(* CODESYS project Flags.library
   Company: _
   DefaultNamespace: Flags
   Title: Flags
   Placeholder: _Flags
   Author: Krystian Lis et al.
   Description: Boolean flags to share between domains.
   Version: 1.0.0

Project tree, tasks and I/O mapping:
  libraries: Debug, * (_); Results, * (_); Strings, * (_); Tags, * (_); Utils, * (_); Tc2_Standard, * (Beckhoff Automation GmbH); Tc2_System, * (Beckhoff Automation GmbH)
  Flag/
    Find/
      function FindFlag [ST]
      function FindManyFlags [ST]
      function FindWcdFlag [ST]
    Flag/
      function block A_Flag [ST]: FB_init
      global variables CFLAG
      function block Flag [ST]: FB_init, IsLowered, IsRised, Lower, Rise, Tag
      interface I_Flag: IsLowered, IsRised, Tag
    List/
      function block FlagList [ST]: _GetByTagIfTagged, _GetByTagIfUntagged, GetByPos, GetByTag, GetExtender, Release, Cap, IsReleased, Length, _ExtendIfTagged, _ExtendIfUntagged, _ExtendIfUntaggedIfNotEmpty, _PushIfTagged, _PushIfUntagged, Extend, Push
      function block FlagListExtender [ST]: List
      interface I_FlagList: GetByPos, GetByTag, GetExtender, Release, Cap, IsReleased, Length
      interface I_MutFlagList: Extend, Push
*)

// Flag/Flag/CFLAG
{attribute 'qualified_only'}
VAR_GLOBAL CONSTANT
	RISED		: Strings.Str := 'Rised';
	LOWERED		: Strings.Str := 'Lowered';
END_VAR

// Flag/Find/FindFlag
FUNCTION FindFlag : Results.Result
VAR_INPUT
	iFlagList		: I_FlagList;
	sToFind			: Strings.Str;
END_VAR
VAR_OUTPUT
	iFlag			: I_Flag;
END_VAR
VAR
	i			: Utils.GenIter(0);
	cmp			: Tags.TagCmp;
END_VAR

IF iFlagList = 0 THEN
	FindFlag := Results.Err.Itf0;
	RETURN;
END_IF

WHILE Results.IsOk(iFlagList.GetByPos(i.Next(), iFlag => iFlag)) DO
	IF cmp.Set(iFlag.Tag).MatchId(sToFind).IsTrue() THEN
		FindFlag := Results.Ok;
		RETURN;
	END_IF
END_WHILE

FindFlag := Results.Err.NoMatch;

END_FUNCTION

// Flag/List/I_FlagList
INTERFACE I_FlagList EXTENDS Debug.I_Debug

METHOD GetByPos : Results.Result
VAR_INPUT
	nPos			: UDINT;
END_VAR
VAR_OUTPUT
	iFlag			: I_Flag;
END_VAR
END_METHOD

METHOD GetByTag : Results.Result
VAR_INPUT
	iTag			: Tags.I_Tag;
END_VAR
VAR_OUTPUT
	iFlag			: I_Flag;
	nPos			: UDINT;
END_VAR
END_METHOD

METHOD GetExtender : FlagListExtender
VAR_INPUT
END_VAR
END_METHOD

METHOD Release : FlagListExtender;
END_METHOD

METHOD Cap : UDINT
VAR_INPUT
END_VAR
END_METHOD

METHOD IsReleased : BOOL
VAR_INPUT
END_VAR
END_METHOD

METHOD Length : UDINT
VAR_INPUT
END_VAR
END_METHOD

END_INTERFACE

// Flag/Flag/I_Flag
INTERFACE I_Flag EXTENDS Debug.I_Debug, Tags.I_Tagged

METHOD IsLowered : BOOL
VAR_INPUT
END_VAR
END_METHOD

METHOD IsRised : BOOL
VAR_INPUT
END_VAR
END_METHOD

PROPERTY Tag : Tags.I_Tag
GET
END_GET
END_PROPERTY

END_INTERFACE

// Flag/List/FlagListExtender
FUNCTION_BLOCK INTERNAL FlagListExtender
VAR
	_iList		: I_FlagList;
END_VAR

PROPERTY INTERNAL List : I_FlagList
GET
List := _iList;
END_GET
SET
_iList := List;
END_SET
END_PROPERTY

END_FUNCTION_BLOCK

// Flag/Find/FindManyFlags
FUNCTION FindManyFlags : Results.Result
VAR_INPUT
	iFlagList		: I_FlagList;
	nResultPou		: ANY;
END_VAR
VAR_IN_OUT
	sToFind		: ARRAY[*] OF Strings.Str;
END_VAR
VAR
	i			: Utils.GenIter(0);
	j			: UDINT;
	cmp			: Tags.TagCmp;
	_iFlag		: I_Flag;
	_nLow		: UDINT := DINT_TO_UDINT(LOWER_BOUND(sToFind, 1));
	_nUp		: UDINT := DINT_TO_UDINT(UPPER_BOUND(sToFind, 1));
	_nResSize	: UDINT := DINT_TO_UDINT(nResultPou.diSize);
	_nExpLen	: UDINT := _nUp - _nLow + 1;
	_nExpSize	: UDINT := _nExpLen * SIZEOF(__UXINT);
	
	_nFound		: UDINT := 0;
END_VAR

IF iFlagList = 0 THEN
	FindManyFlags := Results.Err.Itf0;
	RETURN;
END_IF

// Ensure lower bound starts at zero
IF _nLow <> 0 THEN
	FindManyFlags := Results.Err.Ovf;
	RETURN;
END_IF

// Ensure result size matches expected size
IF _nResSize <> _nExpSize THEN
	FindManyFlags := Results.Err.NoMatch;
	RETURN;
END_IF

// Check if result pointer is null
IF nResultPou.pValue = 0 THEN
	FindManyFlags := Results.Err.Ptr0;
	RETURN;
END_IF

// Iterate over the flag list
WHILE Results.IsOk(iFlagList.GetByPos(i.Next(), iFlag => _iFlag)) DO
	cmp.Set(_iFlag.Tag);
	FOR j := _nLow TO _nUp DO
		// Match the string and copy if successful
		IF cmp.MatchId(sToFind[j]).IsTrue() THEN
			Tc2_System.MEMCPY(ADR(nResultPou.pValue) + SIZEOF(__UXINT) * j, ADR(_iFlag), SIZEOF(__UXINT));
			_nFound := _nFound + 1;
			sToFind[j] := '';  // Mark as found
			EXIT;  // Break after first match (since there should be only one)
		END_IF
	END_FOR;
	
	// Early exit if all entries are found (this condition can be removed if only one flag is expected)
	IF _nFound = (_nUp - _nLow + 1) THEN
		FindManyFlags := Results.Ok;
		RETURN;
	END_IF 
END_WHILE

// Final check to see if all entries were processed
FOR j := _nLow TO _nUp DO
	IF sToFind[j] <> '' THEN  // Check for unfound entries
		FindManyFlags := Results.Err.Udf;  // Error if any remain unfound (handled at higher level)
		RETURN;
	END_IF
END_FOR

// Return success if everything is found
FindManyFlags := Results.Ok;

END_FUNCTION

// Flag/Flag/Flag
FUNCTION_BLOCK Flag IMPLEMENTS I_Flag
VAR
	_fbTag				: Tags.Tag;
	_bState				: BOOL;
END_VAR

//FB_Init is always available implicitly and it is used primarily for initialization.
//The return value is not evaluated. For a specific influence, you can also declare the
//methods explicitly and provide additional code there with the standard initialization
//code. You can evaluate the return value.
METHOD FB_Init: BOOL
VAR_INPUT
    bInitRetains: BOOL; // TRUE: the retain variables are initialized (reset warm / reset cold)
    bInCopyCode: BOOL;  // TRUE: the instance will be copied to the copy code afterward (online change)  
END_VAR
_fbTag.Option := CFLAG.LOWERED;
END_METHOD

METHOD IsLowered : BOOL
VAR_INPUT
END_VAR
IsLowered := _bState = FALSE;
END_METHOD

METHOD IsRised : BOOL
VAR_INPUT
END_VAR
IsRised := _bState = TRUE;
END_METHOD

METHOD Lower : BOOL
VAR_INPUT
END_VAR
_bState := FALSE;
_fbTag.Option := CFLAG.LOWERED;
END_METHOD

METHOD Rise : BOOL
VAR_INPUT
END_VAR
_bState := TRUE;
_fbTag.Option := CFLAG.RISED;
END_METHOD

PROPERTY Tag : Tags.I_Tag
GET
Tag := _fbTag;
END_GET
END_PROPERTY

END_FUNCTION_BLOCK

// Flag/Find/FindWcdFlag
FUNCTION FindWcdFlag : Results.Result
VAR_INPUT
	iFlagList		: I_FlagList;
	sToFind			: Strings.Str;
END_VAR
VAR_OUTPUT
	iFlag			: I_Flag;
END_VAR
VAR
	i			: Utils.GenIter(0);
	cmp			: Tags.TagCmp;
END_VAR

IF iFlagList = 0 THEN
	FindWcdFlag := Results.Err.Itf0;
	RETURN;
END_IF

WHILE Results.IsOk(iFlagList.GetByPos(i.Next(), iFlag => iFlag)) DO
	IF cmp.Set(iFlag.Tag).MatchWcdId(sToFind).IsTrue() THEN
		FindWcdFlag := Results.Ok;
		RETURN;
	END_IF
END_WHILE

FindWcdFlag := Results.Err.NoMatch;

END_FUNCTION

// Flag/Flag/A_Flag
FUNCTION_BLOCK A_Flag IMPLEMENTS Debug.I_Debug;

//FB_Init is always available implicitly and it is used primarily for initialization.
//The return value is not evaluated. For a specific influence, you can also declare the
//methods explicitly and provide additional code there with the standard initialization
//code. You can evaluate the return value.
METHOD FB_Init: BOOL
VAR_INPUT
    bInitRetains: BOOL; // TRUE: the retain variables are initialized (reset warm / reset cold)
    bInCopyCode: BOOL;  // TRUE: the instance will be copied to the copy code afterward (online change)
	iFlagList				: I_MutFlagList;
	iFlag					: I_Flag;
END_VAR
IF iFlagList = 0 THEN
	Debug.DebugMsg(THIS^, ': iFlagList: Itf = 0!');
	RETURN;
END_IF
IF iFlag = 0 THEN
	Debug.DebugMsg(THIS^, ': iFlag: Itf = 0!');
	RETURN;
END_IF

CASE iFlagList.Push(iFlag) OF
	Results.Ok:
		// No Error
	Results.None:
		Debug.DebugMsg(iFlagList, Tc2_Standard.CONCAT(__POUNAME(), ': Tried to insert a double!'));
		Debug.DebugMsg(iFlag, 'Im a double!');
	Results.Err.Ovf:
		Debug.DebugMsg(iFlagList, Tc2_Standard.CONCAT(__POUNAME(), ': Overflow!'));
		Debug.DebugMsg(iFlag, 'Cause of overflow!');
	Results.Err.NoMatch:
		Debug.DebugMsg(iFlagList, Tc2_Standard.CONCAT(__POUNAME(), ': No Match!'));
		Debug.DebugMsg(iFlag, 'This already have an owner!');
	ELSE
		Debug.DebugMsg(iFlagList, Tc2_Standard.CONCAT(__POUNAME(), ': Unknown Error!'));
		Debug.DebugMsg(iFlag, 'Cause!');		
END_CASE
END_METHOD

END_FUNCTION_BLOCK

// Flag/List/I_MutFlagList
INTERFACE I_MutFlagList EXTENDS Debug.I_Debug, I_FlagList

METHOD Extend 			: Results.Result
VAR_INPUT
	fbFlagListExtend	: FlagListExtender;
END_VAR
END_METHOD

METHOD Push : Results.Result
VAR_INPUT
	iFlag			: I_Flag;
END_VAR
VAR_OUTPUT
	nPos			: UDINT;
END_VAR
END_METHOD

END_INTERFACE

// Flag/List/FlagList
FUNCTION_BLOCK FlagList
VAR_GENERIC CONSTANT
	nMax				: UDINT(0..16#FFFFFFE) := 1;
END_VAR
IMPLEMENTS I_FlagList, I_MutFlagList
VAR
	_bIsReleased		: BOOL;
	_iFlag				: ARRAY[0..nMax] OF I_Flag;
	_nLen				: UDINT;
	_fbTagOwner			: Tags.TagOwner;
END_VAR

METHOD PRIVATE _GetByTagIfTagged : Results.Result
VAR_INPUT
	iTag				: Tags.I_Tag;
END_VAR
VAR_OUTPUT
	iFlag				: I_Flag;
	nPos				: UDINT;
END_VAR
IF iTag.Owner <> _fbTagOwner.Self THEN
	_GetByTagIfTagged := Results.None;
	RETURN;
END_IF

iFlag := _iFlag[iTag.Cache];
_GetByTagIfTagged := Results.Ok;
nPos := iTag.Cache;
END_METHOD

METHOD PRIVATE _GetByTagIfUntagged : Results.Result
VAR_INPUT
	iTag				: Tags.I_Tag;
END_VAR
VAR_OUTPUT
	iFlag				: I_Flag;
	nPos				: UDINT;
END_VAR
VAR
	i					: UDINT;
	cmp					: Tags.TagCmp;
END_VAR
FOR i := 0 TO _nLen - 1 DO
	IF cmp.Set(iTag).Match(_iFlag[i].Tag).IsTrue() THEN
		_GetByTagIfUntagged := Results.Ok;
		RETURN;
	END_IF	
END_FOR
END_METHOD

METHOD GetByPos : Results.Result
VAR_INPUT
	nPos		: UDINT;
END_VAR
VAR_OUTPUT
	iFlag		: I_Flag;
END_VAR
IF nPos > nMax THEN
	GetByPos := Results.Err.Ovf;
	RETURN;
END_IF

iFlag := _iFlag[nPos];
IF iFlag <> 0 THEN
	GetByPos := Results.Ok;
END_IF
END_METHOD

METHOD GetByTag : Results.Result;
VAR_INPUT
	iTag				: Tags.I_Tag;
END_VAR
VAR_OUTPUT
	iFlag				: I_Flag;
	nPos				: UDINT;
END_VAR
IF _nLen = 0 THEN
	GetByTag := Results.None;
	RETURN;
END_IF

IF iTag = 0 THEN
	GetByTag := Results.Err.Itf0;
	RETURN;
END_IF

IF _bIsReleased THEN
	GetByTag := _GetByTagIfUntagged(iTag, iFlag => iFlag, nPos => nPos);
ELSE
	GetByTag := _GetByTagIfTagged(iTag, iFlag => iFlag, nPos => nPos);
END_IF
END_METHOD

METHOD GetExtender : FlagListExtender
VAR_INPUT
END_VAR
GetExtender.List := THIS^;
END_METHOD

METHOD Release 				: FlagListExtender;
VAR
	i						: UDINT;
END_VAR
IF NOT _bIsReleased THEN
	FOR i := 0 TO _nLen - 1 DO
		_iFlag[i].Tag.Leave(_fbTagOwner);
	END_FOR
	
	_bIsReleased := TRUE;
END_IF

Release.List := THIS^;
END_METHOD

METHOD Cap : UDINT
VAR_INPUT
END_VAR
Cap := nMax;
END_METHOD

METHOD IsReleased : BOOL
VAR_INPUT
END_VAR
IsReleased := _bIsReleased;
END_METHOD

METHOD Length : UDINT
VAR_INPUT
END_VAR
Length := _nLen;
END_METHOD

METHOD PRIVATE _ExtendIfTagged : Results.Result
VAR_INPUT
	iFlagList			: I_FlagList;
END_VAR
VAR
	i					: UDINT;
	_iExtFlag			: I_Flag;
END_VAR
IF NOT iFlagList.IsReleased() THEN
	_ExtendIfTagged := Results.Err.NoMatch;
	RETURN;
END_IF

IF iFlagList.Length() + _nLen > nMax THEN
	_ExtendIfTagged := Results.Err.Ovf;
	RETURN;
END_IF

WHILE Results.IsOk(iFlagList.GetByPos(i, iFlag => _iExtFlag)) DO
	i := i + 1;
	_iExtFlag.Tag.Join(_fbTagOwner, _nLen);
	_iFlag[_nLen] := _iExtFlag;
	_nLen := _nLen + 1;
END_WHILE

_ExtendIfTagged := Results.Ok;
END_METHOD

METHOD PRIVATE _ExtendIfUntagged : Results.Result
VAR_INPUT
	iFlagList			: I_FlagList;
END_VAR
VAR
	i					: UDINT;
	j					: UDINT;

	_iExtFlag			: I_Flag;
	
END_VAR
IF _nLen <> 0 THEN
	_ExtendIfUntagged := _ExtendIfUntaggedIfNotEmpty(iFlagList);
ELSE
	IF iFlagList.Cap() > nMax THEN
		_ExtendIfUntagged := Results.Err.Ovf;
		RETURN;
	END_IF	

	WHILE Results.IsOk(iFlagList.GetByPos(i, iFlag => _iExtFlag)) DO
		i := i + 1;
		_iExtFlag.Tag.Join(_fbTagOwner, _nLen);
		_iFlag[_nLen] := _iExtFlag;
		_nLen := _nLen + 1;
	END_WHILE
	
	_ExtendIfUntagged := Results.Ok;
END_IF
END_METHOD

METHOD PRIVATE _ExtendIfUntaggedIfNotEmpty : Results.Result
VAR_INPUT
	iFlagList			: I_FlagList;
END_VAR
VAR
	i					: UDINT;
	j					: UDINT;
	k					: UDINT;

	_iTemp				: ARRAY[0..nMax] OF I_Flag;

	_nExtLen			: UDINT;
	_iExtFlag			: I_Flag;
END_VAR
WHILE Results.IsOk(iFlagList.GetByPos(i, iFlag => _iExtFlag)) DO
	
	FOR j := 0 TO _nLen - 1 DO
		IF _iFlag[j] = _iExtFlag THEN
			_iExtFlag := 0;
			EXIT;
		END_IF	
	END_FOR
	
	IF _iExtFlag <> 0 THEN
		_iTemp[k] := _iExtFlag;
		k := k + 1;
	END_IF
	
	i := i + 1;
END_WHILE

IF k = 0 THEN
	_ExtendIfUntaggedIfNotEmpty := Results.Ok;
	RETURN;
END_IF

FOR i := 0 TO k - 1 DO
	_iFlag[_nLen] := _iTemp[i];
	_nLen := _nLen + 1;
END_FOR

_ExtendIfUntaggedIfNotEmpty := Results.Ok;
END_METHOD

METHOD PRIVATE _PushIfTagged : Results.Result
VAR_INPUT
	iFlag			: I_Flag;
END_VAR
VAR_OUTPUT
	nPos			: UDINT;
END_VAR
VAR
	_iTag			: Tags.I_Tag;
END_VAR
IF iFlag = 0 THEN
	_PushIfTagged := Results.Err.Itf0;
	RETURN;
END_IF

IF nMax < _nLen THEN
	_PushIfTagged := Results.Err.Ovf;
	RETURN;
END_IF

IF Results.IsErr(iFlag.Tag.Join(_fbTagOwner, _nLen), eCarry => _PushIfTagged) THEN
	RETURN;
END_IF

_iFlag[_nLen] := iFlag;
_nLen := _nLen + 1;
END_METHOD

METHOD PRIVATE _PushIfUntagged : Results.Result
VAR_INPUT
	iFlag			: I_Flag;
END_VAR
VAR_OUTPUT
	nPos			: UDINT;
END_VAR
VAR
	i				: UDINT;
END_VAR
IF iFlag = 0 THEN
	_PushIfUntagged := Results.Err.Itf0;
	RETURN;
END_IF

IF nMax < _nLen THEN
	_PushIfUntagged := Results.Err.Ovf;
	RETURN;
END_IF

FOR i := 0 TO _nLen - 1 DO
	IF _iFlag[i] = iFlag THEN
		_PushIfUntagged := Results.None;
		RETURN;
	END_IF	
END_FOR

_iFlag[_nLen] := iFlag;
_nLen := _nLen + 1;
_PushIfUntagged := Results.Ok;
END_METHOD

METHOD Extend 			: Results.Result
VAR_INPUT
	fbFlagListExtend	: FlagListExtender;
END_VAR
VAR
	_iFlagList			: I_FlagList;
	_iThis				: I_FlagList := THIS^;
END_VAR
_iFlagList := fbFlagListExtend.List;

IF _iFlagList = 0 THEN
	Extend := Results.Err.Itf0;
	RETURN;
END_IF

IF _iFlagList = _iThis THEN
	Extend := Results.Err.ItfEq;
	RETURN;
END_IF


IF _bIsReleased THEN
	Extend :=_ExtendIfUntagged(_iFlagList);
ELSE
	Extend := _ExtendIfTagged(_iFlagList);
END_IF
END_METHOD

METHOD Push : Results.Result
VAR_INPUT
	iFlag			: I_Flag;
END_VAR
VAR_OUTPUT
	nPos			: UDINT;
END_VAR
IF _bIsReleased THEN
	Push :=_PushIfuntagged(iFlag, nPos => nPos);
ELSE
	Push := _PushIfTagged(iFlag, nPos => nPos);
END_IF
END_METHOD

END_FUNCTION_BLOCK
